// TIA Portal V17 export
// export: Created 2022-07-28T18:02:50.7738126Z, ExportSetting None, DisplayName Totally Integrated Automation Portal, DisplayVersion V17, DisplayName TIA Portal Openness, DisplayVersion V17, DisplayName TIA Portal Teamcenter Gateway, DisplayVersion V17, DisplayName TIA Portal Version Control Interface, DisplayVersion V17, DisplayName TIA Portal Test Suite Advanced, DisplayVersion V17, DisplayName SINAMICS Startdrive Advanced, DisplayVersion V17, DisplayName SINAMICS DCC, DisplayVersion V17, DisplayName SINAMICS Startdrive G130, G150, S120, S150, SINAMICS MV, S210, DisplayVersion V17, DisplayName SINAMICS Startdrive G110M, G120, G120C, G120D, G120P, G115D, DisplayVersion V17, DisplayName STEP 7 Professional, DisplayVersion V17, DisplayName SIMATIC Energy Suite, DisplayVersion V17, DisplayName STEP 7 CFC, DisplayVersion V17, DisplayName STEP 7 Safety, DisplayVersion V17, DisplayName WinCC Advanced / Unified PC, DisplayVersion V17, DisplayName SIMATIC Visualization Architect, DisplayVersion V17
FUNCTION_BLOCK "lib_fb_TurningSensor"   // FB14, SCL
{ S7_Optimized_Access := 'TRUE' }
// stored: MemoryReserve 100, SetENOAutomatically false
   VAR_INPUT
      iSensorSignal : Bool;   // Signal from sensor input
      iStartCmd : Bool;   // Run command has been set
      iiSensorType : Int;   // 0 - disabled; 1 - descrete signal; 2 - pulses when rotating
      irCycleTime : Real;   // Last cycle tyme, msec
      irMaxPulsesDelay : Real := 1.0;   // Max delay between pulses (for type 1 sensor), sec
      irMaxStartTime : Real := 5.0;   // Max Delay between motor start command and shaft rotation, sec
      irMaxStopTime : Real := 5.0;   // Max Delay between motor and shaft stoping, sec
   END_VAR
   VAR_OUTPUT
      oResult : Bool;   // TRUE if shaft rotates
      oStartAlarm : Bool;   // Start time exceeded
      oStopAlarm : Bool;   // Start time exceeded
   END_VAR
   VAR
      sdb_InputPulse : "Lib_FB_Edge";
      sdb_TOF_Pulses : "Lib_FB_Timer_OFF_Simple";   // If false, then the shaft is stopped
      sdb_TON_StartDelay : "Lib_FB_Timer_ON_Simple";   // Delay while not rotating after start command. If true, then fault
      sdb_TON_StopDelay : "Lib_FB_Timer_ON_Simple";   // Delay while rotating after stop command. If true, then fault
   END_VAR
   VAR_TEMP
      tb_ShaftRotates : Bool;
      tb_EnableOuts : Bool;   // 1 - enabled, 0 - disabled
   END_VAR
BEGIN


   //  Check sensor type
   CASE #iiSensorType OF
       1:  // Descrete signal
           #tb_ShaftRotates := #iSensorSignal;
           #tb_EnableOuts := true;
       2:  // Pulses when rotating
           #sdb_InputPulse.IB_Input := #iSensorSignal;

           #sdb_InputPulse();

           #sdb_TOF_Pulses.IB_StartTimerInput := #sdb_InputPulse.QB_EdgePos;
           #sdb_TOF_Pulses.IR_SpTime := #irMaxPulsesDelay;
           #sdb_TOF_Pulses.IR_CycleTime := #irCycleTime;

           #sdb_TOF_Pulses();

           #tb_ShaftRotates := #sdb_TOF_Pulses.QB_TimerOut;
           #tb_EnableOuts := true;
       ELSE
           #tb_EnableOuts := false;
   END_CASE;

   #sdb_TON_StartDelay(IB_StartTimerInput := (#iStartCmd AND NOT #tb_ShaftRotates) AND #tb_EnableOuts,
                       IR_CycleTime := #irCycleTime,
                       IR_SpTime := #irMaxStartTime);

   #sdb_TON_StopDelay(IB_StartTimerInput := (NOT #iStartCmd AND #tb_ShaftRotates) AND #tb_EnableOuts,
                      IR_CycleTime := #irCycleTime,
                      IR_SpTime := #irMaxStopTime);



   //  Alarms
   #oStartAlarm := #sdb_TON_StartDelay.QB_TimerOut;
   #oStopAlarm := #sdb_TON_StopDelay.QB_TimerOut;
   //  Status
   #oResult := #tb_ShaftRotates AND #tb_EnableOuts;
END_FUNCTION_BLOCK
